(* IEC 61131-3 sources: 2026_Projet_YGO_ExcavatriceDragage/CODE/SIMULATION/PLC_TESTS/CORE, 4 files *)

(* ---- FB_TestSequencer.st ---- *)
FUNCTION_BLOCK FB_TestSequencer
VAR_INPUT
    Start       : BOOL;              // Front : lance à FirstStepId
    Abort       : BOOL;              // Niveau : arrêt immédiat propre
    FirstStepId : INT;               // Run all = 1er SETUP ; run one = FirstStep du case visé
END_VAR
VAR_IN_OUT                           // 🔗 zéro copie
    StepTable      : ARRAY[1..GVL_PLC_Tests_Const.MaxSteps]      OF ST_TestStepConfig;
    CheckTable     : ARRAY[1..GVL_PLC_Tests_Const.MaxChecks]     OF ST_TestCheckConfig;
    CaseTable      : ARRAY[1..GVL_PLC_Tests_Const.MaxTestCases]  OF ST_TestCaseConfig;
    InvariantTable : ARRAY[1..GVL_PLC_Tests_Const.MaxInvariants] OF ST_TestInvariantConfig;
    ProbeBool      : ARRAY[1..GVL_PLC_Tests_Const.MaxProbeBool]  OF BOOL;
    ProbeDint      : ARRAY[1..GVL_PLC_Tests_Const.MaxProbeDint]  OF DINT;
    ProbeReal      : ARRAY[1..GVL_PLC_Tests_Const.MaxProbeReal]  OF REAL;
    Report         : ST_TestSuiteReport;
END_VAR
VAR_OUTPUT
    Busy                : BOOL;
    Done                : BOOL;
    AnyFailed           : BOOL;
    ConfigError         : BOOL;      // 🔒 Table invalide -> refus de lancer
    ConfigErrorStepId   : INT;
    ConfigErrorCheckIdx : INT;
    CurrentStepId       : INT;
    ActiveStimulusId    : INT;       // ⚡ consommé par le domaine
    StepElapsed         : TIME;      // Pour l'IHM
END_VAR
VAR
    StartTrig           : R_TRIG;
    StepTimer           : TON;
    DwellTimer          : TON;
    Checks              : ARRAY[1..GVL_PLC_Tests_Const.MaxChecksPerStep] OF FB_TestCheck;
    InvChecks           : ARRAY[1..GVL_PLC_Tests_Const.MaxInvariants]    OF FB_TestCheck;
    InvArmed            : ARRAY[1..GVL_PLC_Tests_Const.MaxInvariants]    OF BOOL;

    // Variables de contrôle internes
    StepStarted         : BOOL;
    CurrentCaseId       : INT;
    Idx                 : INT;
    Jdx                 : INT;
    Kdx                 : INT;
    Valid               : BOOL;

    // 🔧 REX : locaux remontés depuis des blocs VAR imbriqués dans le corps
    AllChecksPassed     : BOOL;
    AnyCheckFailed      : BOOL;
    FailedCheckIdxLocal : INT;
    FailReasonLocal     : E_TestFailReason;
    ObsBoolLocal        : BOOL;
    ObsDintLocal        : DINT;
    ObsRealLocal        : REAL;
    NeverDuringPassed   : BOOL;
    SuiteAllPassed      : BOOL;
    FirstFailedCase     : INT;
    CaseIdx             : INT;
    CaseStartStep       : INT;
    CaseStep            : INT;
    CaseOk              : BOOL;
    CaseExecuted        : BOOL;
    CaseFailedStep      : INT;
    CaseDuration        : TIME;
    CaseFailReason      : E_TestFailReason;
END_VAR
// === IMPLEMENTATION ===
StartTrig(CLK := Start);

// 1. Validation de la configuration sur front de Start
IF StartTrig.Q THEN
    ConfigError := FALSE;
    ConfigErrorStepId := 0;
    ConfigErrorCheckIdx := 0;

    // Validation des étapes
    FOR Idx := 1 TO GVL_PLC_Tests_Const.MaxSteps DO
        IF StepTable[Idx].CaseId > 0 THEN
            // Vérification des NextOn
            IF StepTable[Idx].NextOnPass < 0 OR StepTable[Idx].NextOnPass > GVL_PLC_Tests_Const.MaxSteps THEN
                ConfigError := TRUE;
                ConfigErrorStepId := Idx;
            ELSIF StepTable[Idx].NextOnFail < 0 OR StepTable[Idx].NextOnFail > GVL_PLC_Tests_Const.MaxSteps THEN
                ConfigError := TRUE;
                ConfigErrorStepId := Idx;
            END_IF;

            // Vérification du Timeout
            IF StepTable[Idx].TimeoutPT <= T#0s THEN
                // Sauf si tous les checks de cette étape sont NEVER_DURING, mais restons stricts : TimeoutPT requis
                ConfigError := TRUE;
                ConfigErrorStepId := Idx;
            END_IF;

            // Vérification des Checks indexés par l'étape
            FOR Jdx := 1 TO GVL_PLC_Tests_Const.MaxChecksPerStep DO
                Kdx := StepTable[Idx].CheckIdx[Jdx];
                IF Kdx > 0 THEN
                    IF Kdx > GVL_PLC_Tests_Const.MaxChecks THEN
                        ConfigError := TRUE;
                        ConfigErrorStepId := Idx;
                        ConfigErrorCheckIdx := Kdx;
                    ELSE
                        // Validation de la sonde associée au check
                        CASE CheckTable[Kdx].Kind OF
                            E_TestCheckKind.BOOL_EQUAL, E_TestCheckKind.BOOL_RISING, E_TestCheckKind.BOOL_FALLING:
                                IF CheckTable[Kdx].ProbeIdx < 1 OR CheckTable[Kdx].ProbeIdx > GVL_PLC_Tests_Const.MaxProbeBool THEN
                                    ConfigError := TRUE;
                                    ConfigErrorStepId := Idx;
                                    ConfigErrorCheckIdx := Kdx;
                                END_IF;
                            E_TestCheckKind.DINT_EQUAL, E_TestCheckKind.DINT_NOT_EQUAL, E_TestCheckKind.DINT_IN_RANGE,
                            E_TestCheckKind.WORD_MASK_ALL, E_TestCheckKind.WORD_MASK_ANY, E_TestCheckKind.WORD_MASK_NONE:
                                IF CheckTable[Kdx].ProbeIdx < 1 OR CheckTable[Kdx].ProbeIdx > GVL_PLC_Tests_Const.MaxProbeDint THEN
                                    ConfigError := TRUE;
                                    ConfigErrorStepId := Idx;
                                    ConfigErrorCheckIdx := Kdx;
                                END_IF;
                            E_TestCheckKind.REAL_IN_RANGE:
                                IF CheckTable[Kdx].ProbeIdx < 1 OR CheckTable[Kdx].ProbeIdx > GVL_PLC_Tests_Const.MaxProbeReal THEN
                                    ConfigError := TRUE;
                                    ConfigErrorStepId := Idx;
                                    ConfigErrorCheckIdx := Kdx;
                                END_IF;
                        END_CASE;
                    END_IF;
                END_IF;
            END_FOR;
        END_IF;
    END_FOR;

    // Si erreur de config, on bloque le démarrage
    IF ConfigError THEN
        RETURN;
    END_IF;
END_IF;

// 2. Abort (Niveau, priorité absolue)
IF Abort THEN
    IF Busy THEN
        Report.InProgress := FALSE;
        Report.Aborted := TRUE;
        Report.AnyFailed := TRUE;

        // Enregistrement de l'échec de l'étape courante
        IF CurrentStepId >= 1 AND CurrentStepId <= GVL_PLC_Tests_Const.MaxSteps THEN
            Report.Steps[CurrentStepId].Executed := TRUE;
            Report.Steps[CurrentStepId].Passed := FALSE;
            Report.Steps[CurrentStepId].FailReason := E_TestFailReason.FAIL_ABORTED;
            Report.Steps[CurrentStepId].Duration := StepElapsed;
        END_IF;

        // Échec du cas de test en cours
        IF CurrentCaseId >= 1 AND CurrentCaseId <= GVL_PLC_Tests_Const.MaxTestCases THEN
            Report.Cases[CurrentCaseId].Ok := FALSE;
            Report.Cases[CurrentCaseId].FailReason := E_TestFailReason.FAIL_ABORTED;
        END_IF;

        Busy := FALSE;
        Done := TRUE;
        AnyFailed := TRUE;
    END_IF;
    ActiveStimulusId := 0;
    StepStarted := FALSE;
    RETURN;
END_IF;

// 3. Démarrage de la suite
IF StartTrig.Q AND NOT ConfigError THEN
    Busy := TRUE;
    Done := FALSE;
    AnyFailed := FALSE;
    CurrentStepId := FirstStepId;
    StepStarted := FALSE;

    // RAZ Rapport
    Report.InProgress := TRUE;
    Report.AllPassed := FALSE;
    Report.AnyFailed := FALSE;
    Report.Aborted := FALSE;
    Report.FailedTestCase := 0;
    Report.CurrentStepId := FirstStepId;
    IF CurrentStepId >= 1 AND CurrentStepId <= GVL_PLC_Tests_Const.MaxSteps THEN
        Report.CurrentCaseId := StepTable[CurrentStepId].CaseId;
    ELSE
        Report.CurrentCaseId := 0;
    END_IF;
    Report.Duration := T#0s;
    Report.RunCounter := Report.RunCounter + 1;

    FOR Idx := 1 TO GVL_PLC_Tests_Const.MaxSteps DO
        Report.Steps[Idx].Executed := FALSE;
        Report.Steps[Idx].Passed := FALSE;
        Report.Steps[Idx].FailReason := E_TestFailReason.FAIL_NONE;
        Report.Steps[Idx].FailedCheckIdx := 0;
        Report.Steps[Idx].FailedInvariantId := 0;
        Report.Steps[Idx].Duration := T#0s;
    END_FOR;

    FOR Idx := 1 TO GVL_PLC_Tests_Const.MaxTestCases DO
        Report.Cases[Idx].Executed := FALSE;
        Report.Cases[Idx].Ok := FALSE;
        Report.Cases[Idx].FailedStepId := 0;
        Report.Cases[Idx].FailReason := E_TestFailReason.FAIL_NONE;
        Report.Cases[Idx].Duration := T#0s;
    END_FOR;

    // RAZ Invariants
    FOR Idx := 1 TO GVL_PLC_Tests_Const.MaxInvariants DO
        InvArmed[Idx] := FALSE;
    END_FOR;
END_IF;

// 4. Moteur d'exécution principal
IF Busy THEN
    // Incrément de la durée globale du run
    Report.Duration := Report.Duration + UDINT_TO_TIME(INT_TO_UDINT(GVL_PLC_Tests_Const.TaskCycleMs));

    // Vérification des bornes de l'étape courante
    IF CurrentStepId < 1 OR CurrentStepId > GVL_PLC_Tests_Const.MaxSteps THEN
        Busy := FALSE;
        Done := TRUE;
        ActiveStimulusId := 0;
        RETURN;
    END_IF;

    CurrentCaseId := StepTable[CurrentStepId].CaseId;
    ActiveStimulusId := StepTable[CurrentStepId].StimulusId;
    Report.CurrentStepId := CurrentStepId;
    Report.CurrentCaseId := CurrentCaseId;

    IF NOT StepStarted THEN
        StepStarted := TRUE;
        StepElapsed := T#0s;
        DwellTimer(IN := FALSE);
        StepTimer(IN := FALSE);

        // Gestion de l'armement/désarmement des invariants
        FOR Idx := 1 TO GVL_PLC_Tests_Const.MaxInvariants DO
            IF InvariantTable[Idx].ArmAtStepId = CurrentStepId THEN
                InvArmed[Idx] := TRUE;
            END_IF;
            IF InvariantTable[Idx].DisarmAtStepId = CurrentStepId THEN
                InvArmed[Idx] := FALSE;
            END_IF;
        END_FOR;
    END_IF;

    // Incrément de la durée de l'étape courante
    StepElapsed := StepElapsed + UDINT_TO_TIME(INT_TO_UDINT(GVL_PLC_Tests_Const.TaskCycleMs));

    // 4.1 Évaluation des invariants actifs
    FOR Idx := 1 TO GVL_PLC_Tests_Const.MaxInvariants DO
        IF InvArmed[Idx] THEN
            InvChecks[Idx](Config := InvariantTable[Idx].Check, Evaluate := TRUE, ProbeBool := ProbeBool, ProbeDint := ProbeDint, ProbeReal := ProbeReal);
            IF InvChecks[Idx].Failed THEN
                // Violation d'invariant -> Transition en échec immédiat
                Report.Steps[CurrentStepId].Executed := TRUE;
                Report.Steps[CurrentStepId].Passed := FALSE;
                Report.Steps[CurrentStepId].FailReason := E_TestFailReason.FAIL_INVARIANT;
                Report.Steps[CurrentStepId].FailedInvariantId := Idx;
                Report.Steps[CurrentStepId].Duration := StepElapsed;
                Report.Steps[CurrentStepId].ObservedBool := InvChecks[Idx].ObservedBool;
                Report.Steps[CurrentStepId].ObservedDint := InvChecks[Idx].ObservedDint;
                Report.Steps[CurrentStepId].ObservedReal := InvChecks[Idx].ObservedReal;

                // Désactivation de l'évaluation
                InvChecks[Idx](Config := InvariantTable[Idx].Check, Evaluate := FALSE, ProbeBool := ProbeBool, ProbeDint := ProbeDint, ProbeReal := ProbeReal);

                // Transition
                IF StepTable[CurrentStepId].FailAction = E_TestFailAction.FAIL_ABORT_SUITE THEN
                    Busy := FALSE;
                    Done := TRUE;
                    AnyFailed := TRUE;
                    ActiveStimulusId := 0;
                ELSE
                    CurrentStepId := StepTable[CurrentStepId].NextOnFail;
                    StepStarted := FALSE;
                END_IF;
                RETURN;
            END_IF;
        END_IF;
    END_FOR;

    // 4.2 Gestion de la temporisation de Dwell
    DwellTimer(IN := TRUE, PT := StepTable[CurrentStepId].DwellPT);
    IF NOT DwellTimer.Q THEN
        // En attente du Dwell, pas d'évaluation des checks d'étape
        FOR Jdx := 1 TO GVL_PLC_Tests_Const.MaxChecksPerStep DO
            Checks[Jdx](Evaluate := FALSE, ProbeBool := ProbeBool, ProbeDint := ProbeDint, ProbeReal := ProbeReal);
        END_FOR;
        RETURN;
    END_IF;

    // 4.3 Évaluation des checks d'étape
    AllChecksPassed     := TRUE;
    AnyCheckFailed      := FALSE;
    FailedCheckIdxLocal := 0;
    FailReasonLocal     := E_TestFailReason.FAIL_NONE;
    ObsBoolLocal        := FALSE;
    ObsDintLocal        := 0;
    ObsRealLocal        := 0.0;

    FOR Jdx := 1 TO GVL_PLC_Tests_Const.MaxChecksPerStep DO
        Kdx := StepTable[CurrentStepId].CheckIdx[Jdx];
        IF Kdx > 0 THEN
            Checks[Jdx](Config := CheckTable[Kdx], Evaluate := TRUE, ProbeBool := ProbeBool, ProbeDint := ProbeDint, ProbeReal := ProbeReal);

            IF Checks[Jdx].Failed THEN
                AnyCheckFailed := TRUE;
                FailedCheckIdxLocal := Kdx;
                FailReasonLocal := Checks[Jdx].FailReason;
                ObsBoolLocal := Checks[Jdx].ObservedBool;
                ObsDintLocal := Checks[Jdx].ObservedDint;
                ObsRealLocal := Checks[Jdx].ObservedReal;
            ELSIF Checks[Jdx].Pending THEN
                AllChecksPassed := FALSE;
            END_IF;
        END_IF;
    END_FOR;

    // 4.4 Prise de verdict
    IF AnyCheckFailed THEN
        // Échec sur un check d'étape
        Report.Steps[CurrentStepId].Executed := TRUE;
        Report.Steps[CurrentStepId].Passed := FALSE;
        Report.Steps[CurrentStepId].FailReason := FailReasonLocal;
        Report.Steps[CurrentStepId].FailedCheckIdx := FailedCheckIdxLocal;
        Report.Steps[CurrentStepId].Duration := StepElapsed;
        Report.Steps[CurrentStepId].ObservedBool := ObsBoolLocal;
        Report.Steps[CurrentStepId].ObservedDint := ObsDintLocal;
        Report.Steps[CurrentStepId].ObservedReal := ObsRealLocal;

        // Reset checks
        FOR Jdx := 1 TO GVL_PLC_Tests_Const.MaxChecksPerStep DO
            Checks[Jdx](Evaluate := FALSE, ProbeBool := ProbeBool, ProbeDint := ProbeDint, ProbeReal := ProbeReal);
        END_FOR;

        IF StepTable[CurrentStepId].FailAction = E_TestFailAction.FAIL_ABORT_SUITE THEN
            Busy := FALSE;
            Done := TRUE;
            AnyFailed := TRUE;
            ActiveStimulusId := 0;
        ELSE
            CurrentStepId := StepTable[CurrentStepId].NextOnFail;
            StepStarted := FALSE;
        END_IF;
        RETURN;
    END_IF;

    StepTimer(IN := TRUE, PT := StepTable[CurrentStepId].TimeoutPT);

    IF AllChecksPassed THEN
        // Succès précoce (vérification MinPT)
        IF StepElapsed < StepTable[CurrentStepId].MinPT THEN
            // Réaction trop rapide = Échec
            Report.Steps[CurrentStepId].Executed := TRUE;
            Report.Steps[CurrentStepId].Passed := FALSE;
            Report.Steps[CurrentStepId].FailReason := E_TestFailReason.FAIL_WINDOW_EARLY;
            Report.Steps[CurrentStepId].Duration := StepElapsed;

            // Reset checks
            FOR Jdx := 1 TO GVL_PLC_Tests_Const.MaxChecksPerStep DO
                Checks[Jdx](Evaluate := FALSE, ProbeBool := ProbeBool, ProbeDint := ProbeDint, ProbeReal := ProbeReal);
            END_FOR;

            IF StepTable[CurrentStepId].FailAction = E_TestFailAction.FAIL_ABORT_SUITE THEN
                Busy := FALSE;
                Done := TRUE;
                AnyFailed := TRUE;
                ActiveStimulusId := 0;
            ELSE
                CurrentStepId := StepTable[CurrentStepId].NextOnFail;
                StepStarted := FALSE;
            END_IF;
        ELSE
            // Validation étape OK
            Report.Steps[CurrentStepId].Executed := TRUE;
            Report.Steps[CurrentStepId].Passed := TRUE;
            Report.Steps[CurrentStepId].Duration := StepElapsed;

            // Prendre snapshot du premier check s'il existe
            IF StepTable[CurrentStepId].CheckIdx[1] > 0 THEN
                Report.Steps[CurrentStepId].ObservedBool := Checks[1].ObservedBool;
                Report.Steps[CurrentStepId].ObservedDint := Checks[1].ObservedDint;
                Report.Steps[CurrentStepId].ObservedReal := Checks[1].ObservedReal;
            END_IF;

            // Reset checks
            FOR Jdx := 1 TO GVL_PLC_Tests_Const.MaxChecksPerStep DO
                Checks[Jdx](Evaluate := FALSE, ProbeBool := ProbeBool, ProbeDint := ProbeDint, ProbeReal := ProbeReal);
            END_FOR;

            CurrentStepId := StepTable[CurrentStepId].NextOnPass;
            StepStarted := FALSE;
        END_IF;
        RETURN;
    END_IF;

    // Gestion du timeout d'étape
    IF StepTimer.Q THEN
        // Si timeout expiré, vérifions si des checks NEVER_DURING sont en attente
        NeverDuringPassed := TRUE;
        FOR Jdx := 1 TO GVL_PLC_Tests_Const.MaxChecksPerStep DO
            Kdx := StepTable[CurrentStepId].CheckIdx[Jdx];
            IF Kdx > 0 THEN
                IF CheckTable[Kdx].Mode = E_TestCheckMode.CHECK_NEVER_DURING THEN
                    // Jamais violé pendant toute la fenêtre
                    Checks[Jdx](Evaluate := FALSE, ProbeBool := ProbeBool, ProbeDint := ProbeDint, ProbeReal := ProbeReal);
                ELSE
                    // Les autres modes auraient dû passer avant le timeout
                    NeverDuringPassed := FALSE;
                END_IF;
            END_IF;
        END_FOR;

        IF NeverDuringPassed THEN
            // Succès par non-violation
            Report.Steps[CurrentStepId].Executed := TRUE;
            Report.Steps[CurrentStepId].Passed := TRUE;
            Report.Steps[CurrentStepId].Duration := StepElapsed;

            CurrentStepId := StepTable[CurrentStepId].NextOnPass;
            StepStarted := FALSE;
        ELSE
            // Timeout classique de l'étape
            Report.Steps[CurrentStepId].Executed := TRUE;
            Report.Steps[CurrentStepId].Passed := FALSE;
            Report.Steps[CurrentStepId].FailReason := E_TestFailReason.FAIL_TIMEOUT;
            Report.Steps[CurrentStepId].Duration := StepElapsed;

            IF StepTable[CurrentStepId].FailAction = E_TestFailAction.FAIL_ABORT_SUITE THEN
                Busy := FALSE;
                Done := TRUE;
                AnyFailed := TRUE;
                ActiveStimulusId := 0;
            ELSE
                CurrentStepId := StepTable[CurrentStepId].NextOnFail;
                StepStarted := FALSE;
            END_IF;
        END_IF;

        // Reset checks
        FOR Jdx := 1 TO GVL_PLC_Tests_Const.MaxChecksPerStep DO
            Checks[Jdx](Evaluate := FALSE, ProbeBool := ProbeBool, ProbeDint := ProbeDint, ProbeReal := ProbeReal);
        END_FOR;
    END_IF;
END_IF;

// 5. Agrégation des résultats en fin de suite (CurrentStepId = 0)
IF Busy AND CurrentStepId = 0 THEN
    Busy := FALSE;
    Done := TRUE;
    ActiveStimulusId := 0;
    Report.InProgress := FALSE;

    // Agrégation des cas de test
    SuiteAllPassed  := TRUE;
    FirstFailedCase := 0;

    FOR CaseIdx := 1 TO GVL_PLC_Tests_Const.MaxTestCases DO
        CaseStartStep := CaseTable[CaseIdx].FirstStep;
        IF CaseStartStep > 0 THEN
            CaseOk := TRUE;
            CaseExecuted := FALSE;
            CaseFailedStep := 0;
            CaseDuration := T#0s;
            CaseFailReason := E_TestFailReason.FAIL_NONE;

            // Parcourir la chaîne d'étapes à partir de FirstStep
            CaseStep := CaseStartStep;
            WHILE CaseStep > 0 AND StepTable[CaseStep].CaseId = CaseIdx DO
                IF Report.Steps[CaseStep].Executed THEN
                    CaseExecuted := TRUE;
                    CaseDuration := CaseDuration + Report.Steps[CaseStep].Duration;
                    IF NOT Report.Steps[CaseStep].Passed THEN
                        CaseOk := FALSE;
                        CaseFailedStep := CaseStep;
                        CaseFailReason := Report.Steps[CaseStep].FailReason;
                    END_IF;
                END_IF;

                // Suivre NextOnPass ou NextOnFail selon l'exécution réelle
                IF Report.Steps[CaseStep].Executed AND NOT Report.Steps[CaseStep].Passed THEN
                    CaseStep := StepTable[CaseStep].NextOnFail;
                ELSE
                    CaseStep := StepTable[CaseStep].NextOnPass;
                END_IF;
            END_WHILE;

            Report.Cases[CaseIdx].Executed := CaseExecuted;
            Report.Cases[CaseIdx].Ok := CaseExecuted AND CaseOk;
            Report.Cases[CaseIdx].FailedStepId := CaseFailedStep;
            Report.Cases[CaseIdx].FailReason := CaseFailReason;
            Report.Cases[CaseIdx].Duration := CaseDuration;

            IF CaseExecuted AND NOT CaseOk THEN
                SuiteAllPassed := FALSE;
                IF FirstFailedCase = 0 THEN
                    FirstFailedCase := CaseIdx;
                END_IF;
            END_IF;
        END_IF;
    END_FOR;

    Report.AllPassed := SuiteAllPassed;
    Report.AnyFailed := NOT SuiteAllPassed;
    Report.FailedTestCase := FirstFailedCase;
    AnyFailed := NOT SuiteAllPassed;
END_IF;

(* ---- FB_TranslationTestCleanup.st ---- *)
// ═══════════════════════════════════════════════════════════════
// 🧪 FB_TranslationTestCleanup — Neutralité Translation M3
// ───────────────────────────────────────────────────────────────
// 🎯 Responsabilité UNIQUE : porter le vecteur d'état NEUTRE complet
//    (tous les overrides M3 relâchés, instance isolée FB_Translation
//    au repos). Source de vérité UNIQUE de "neutre" — appelée depuis
//    le fichier suite (SUITE_TRANSLATION/FB_TranslationValidation.st)
//    à la fois dans le CASE stimulus (StimulusId=0) ET, en garantie
//    structurelle indépendante, sur tout chemin où la suite n'est pas
//    Busy (ceinture + bretelles, AF_Partie-14 §7.3.2).
// 🚫 Ne force JAMAIS une sortie de commande calculée — uniquement les
//    surcharges capteurs amont (GVL_PLC_Tests.OverrideM3*) et les
//    entrées de l'instance de test isolée.
// ═══════════════════════════════════════════════════════════════

FUNCTION_BLOCK PUBLIC FB_TranslationTestCleanup
VAR_INPUT
    Apply : BOOL; // TRUE = force la neutralité maintenant
END_VAR
VAR_OUTPUT
    OverrideAtTremie          : BOOL;
    OverrideBrakeStuckOpen    : BOOL;
    OverridePhantomFreq       : BOOL;
    OverrideSensorsWordActive : BOOL;
    UnderTestDirection        : INT;
    UnderTestStartStop        : BOOL;
    UnderTestSlowdownSensor   : BOOL;
    NeutralConfirmed          : BOOL; // TRUE dès que la neutralité a été appliquée ce scan
END_VAR
// === IMPLEMENTATION ===
IF Apply THEN
    OverrideAtTremie := FALSE;
    OverrideBrakeStuckOpen := FALSE;
    OverridePhantomFreq := FALSE;
    OverrideSensorsWordActive := FALSE;
    UnderTestDirection := 0;
    UnderTestStartStop := FALSE;
    UnderTestSlowdownSensor := FALSE;
    NeutralConfirmed := TRUE;
ELSE
    NeutralConfirmed := FALSE;
END_IF;

(* ---- FB_TranslationTestFixture.st ---- *)
// ═══════════════════════════════════════════════════════════════
// 🧪 FB_TranslationTestFixture — Précondition Translation M3
// ───────────────────────────────────────────────────────────────
// 🎯 Responsabilité UNIQUE : décider si un Start est recevable
//    (Niveaux 1/2 de la défense en profondeur, AF_Partie-14 §7.3.3) :
//    simulation active + aucune E/S M3 recâblée réelle. Ne fait AUCUNE
//    attente d'état sain (ça reste la responsabilité de l'étape SETUP
//    de chaque cas, via FB_TranslationStepExecutor — §7.3.5).
// 🔒 Un refus ici est TOUJOURS explicite (PRECONDITION_FAILED),
//    jamais un silence (audit v1.0 C3).
// ═══════════════════════════════════════════════════════════════

FUNCTION_BLOCK PUBLIC FB_TranslationTestFixture
VAR_INPUT
    CheckRequested        : BOOL; // Front : nouvelle vérification demandée (sur Start suite)
    SimulationModeActive  : BOOL;
    SimGateOk             : BOOL; // Niveau 2 : aucune E/S M3 (*IsReal) incompatible
END_VAR
VAR_OUTPUT
    FixturePassed  : BOOL;
    FixtureFailed  : BOOL;
    FailReason     : STRING(120);
END_VAR
VAR
    CheckTrig : R_TRIG;
END_VAR
// === IMPLEMENTATION ===
CheckTrig(CLK := CheckRequested);

IF CheckTrig.Q THEN
    IF NOT SimulationModeActive THEN
        FixturePassed := FALSE;
        FixtureFailed := TRUE;
        FailReason := 'Simulation non active (GVL_Simulation.SimulationModeActive=FALSE)';
    ELSIF NOT SimGateOk THEN
        FixturePassed := FALSE;
        FixtureFailed := TRUE;
        FailReason := 'E/S M3 recablees reelles (*IsReal) incompatibles avec le banc de test';
    ELSE
        FixturePassed := TRUE;
        FixtureFailed := FALSE;
        FailReason := '';
    END_IF;
END_IF;

(* ---- FB_TranslationTestRuntime.st ---- *)
// ═══════════════════════════════════════════════════════════════
// 🧪 FB_TranslationTestRuntime — Cycle de vie protégé Translation M3
// ───────────────────────────────────────────────────────────────
// 🎯 Responsabilité UNIQUE : posséder le lifecycle atomique du run :
//    IDLE → RUN → CLEANUP → WAIT_NEUTRAL → VERIFY → TERMINAL.
// 🔒 Aucun terminal n'est publié avant neutralité confirmée.
// ═══════════════════════════════════════════════════════════════

FUNCTION_BLOCK PUBLIC FB_TranslationTestRuntime
VAR_INPUT
    Start   : BOOL;
    Abort   : BOOL;
    CaseId  : INT;
    PlanConfigError         : BOOL;
    PlanConfigErrorStepId   : INT;
    PlanConfigErrorCheckIdx : INT;
    PlanConfigErrorMessage  : STRING(160);
    SimulationModeActive    : BOOL;
    SimGateOk               : BOOL;
    NeutralConfirmed        : BOOL; // Neutralité réellement appliquée au scan précédent
    WatchdogLimitMs         : DINT := 180000; // Paramétrable pour autotest du framework
    CleanupTimeoutScans     : INT := 20;      // Délai max de confirmation du neutre
END_VAR
VAR_IN_OUT
    StepTable  : ARRAY[1..GVL_PLC_Tests_Const.MaxSteps]      OF ST_TestStepConfig;
    CheckTable : ARRAY[1..GVL_PLC_Tests_Const.MaxChecks]     OF ST_TestCheckConfig;
    CaseTable  : ARRAY[1..GVL_PLC_Tests_Const.MaxTestCases]  OF ST_TestCaseConfig;
    ProbeBool  : ARRAY[1..GVL_PLC_Tests_Const.MaxProbeBool]  OF BOOL;
    ProbeDint  : ARRAY[1..GVL_PLC_Tests_Const.MaxProbeDint]  OF DINT;
    ProbeReal  : ARRAY[1..GVL_PLC_Tests_Const.MaxProbeReal]  OF REAL;
    Report     : ST_TestSuiteReport;
    Result     : ST_TranslationTestResult;
END_VAR
VAR_OUTPUT
    Busy                : BOOL;
    Done                : BOOL;
    AnyFailed           : BOOL;
    ActiveStimulusId    : INT;
    StepElapsed         : TIME;
    TerminalState       : E_TestTerminalState;
    ConfigError         : BOOL;
    ConfigErrorStepId   : INT;
    ConfigErrorCheckIdx : INT;
    ErrorCode           : INT;
    ErrorMessage        : STRING(160);
    StartRejected       : BOOL; // Impulsion : Start reçu hors IDLE/TERMINAL
    CleanupRequest      : BOOL; // Niveau : imposer le vecteur neutre complet
END_VAR
VAR CONSTANT
    RuntimeIdle        : INT := 0;
    RuntimeRun         : INT := 10;
    RuntimeCleanup     : INT := 20;
    RuntimeWaitNeutral : INT := 30;
    RuntimeVerify      : INT := 40;
    RuntimeTerminal    : INT := 50;
END_VAR
VAR
    instFixture   : FB_TranslationTestFixture;
    instExecutor  : FB_TranslationStepExecutor;
    instFinalizer : FB_TranslationReportFinalizer;
    StartTrig     : R_TRIG;
    RuntimeState  : INT := 0;
    ExecutorStart : BOOL;
    ExecutorAbort : BOOL;
    RunStartPulse : BOOL;
    FinalizePulse : BOOL;
    PendingTerminalState : E_TestTerminalState;
    PendingErrorCode     : INT;
    PendingErrorMessage  : STRING(160);
    SuiteElapsed         : TIME;
    NeutralWaitScans     : INT;
    CleanupElapsedScans  : INT;
END_VAR
// === IMPLEMENTATION ===
StartTrig(CLK := Start);
StartRejected := FALSE;
ExecutorStart := FALSE;
ExecutorAbort := FALSE;
RunStartPulse := FALSE;
FinalizePulse := FALSE;
CleanupRequest := (RuntimeState = RuntimeCleanup)
               OR (RuntimeState = RuntimeWaitNeutral)
               OR (RuntimeState = RuntimeVerify);

// 🎮 Un Start pendant un run/cleanup est refusé sans modifier le run actif.
IF StartTrig.Q AND RuntimeState <> RuntimeIdle AND RuntimeState <> RuntimeTerminal THEN
    StartRejected := TRUE;
END_IF;

// 🚪 Fixture appelée CHAQUE scan : son R_TRIG interne est ainsi toujours réarmé.
instFixture(CheckRequested := StartTrig.Q,
            SimulationModeActive := SimulationModeActive,
            SimGateOk := SimGateOk);

// 🟢 Nouveau run accepté depuis IDLE ou TERMINAL.
IF StartTrig.Q AND (RuntimeState = RuntimeIdle OR RuntimeState = RuntimeTerminal) THEN
    RunStartPulse := TRUE;
    Done := FALSE;
    SuiteElapsed := T#0s;
    NeutralWaitScans := 0;
    CleanupElapsedScans := 0;
    PendingTerminalState := E_TestTerminalState.TEST_TERMINAL_NONE;
    PendingErrorCode := 0;
    PendingErrorMessage := '';

    IF PlanConfigError THEN
        PendingTerminalState := E_TestTerminalState.TEST_TERMINAL_CONFIG_ERROR;
        PendingErrorCode := 1002;
        PendingErrorMessage := CONCAT('Table invalide : ', PlanConfigErrorMessage);
        RuntimeState := RuntimeCleanup;
    ELSIF CaseId < 0 OR CaseId > 6 THEN
        PendingTerminalState := E_TestTerminalState.TEST_TERMINAL_CONFIG_ERROR;
        PendingErrorCode := 1001;
        PendingErrorMessage := 'CaseId invalide (attendu 0..6)';
        RuntimeState := RuntimeCleanup;
    ELSIF instFixture.FixtureFailed THEN
        PendingTerminalState := E_TestTerminalState.TEST_TERMINAL_PRECONDITION_FAILED;
        PendingErrorCode := 1010;
        PendingErrorMessage := CONCAT('PRECONDITION_FAILED : ', instFixture.FailReason);
        RuntimeState := RuntimeCleanup;
    ELSE
        ExecutorStart := TRUE;
        RuntimeState := RuntimeRun;
    END_IF;
END_IF;

// 🛡️ Causes de sortie du RUN : watchdog > gate perdue > abort opérateur.
IF RuntimeState = RuntimeRun THEN
    SuiteElapsed := SuiteElapsed + UDINT_TO_TIME(INT_TO_UDINT(GVL_PLC_Tests_Const.TaskCycleMs));
    IF SuiteElapsed >= DINT_TO_TIME(WatchdogLimitMs) THEN
        ExecutorAbort := TRUE;
        PendingTerminalState := E_TestTerminalState.TEST_TERMINAL_WATCHDOG_TIMEOUT;
        PendingErrorCode := 1020;
        PendingErrorMessage := 'Watchdog suite Translation expire';
    ELSIF NOT SimulationModeActive OR NOT SimGateOk THEN
        ExecutorAbort := TRUE;
        PendingTerminalState := E_TestTerminalState.TEST_TERMINAL_PRECONDITION_FAILED;
        PendingErrorCode := 1011;
        PendingErrorMessage := 'Gate Translation perdue pendant le run';
    ELSIF Abort THEN
        ExecutorAbort := TRUE;
        PendingTerminalState := E_TestTerminalState.TEST_TERMINAL_ABORTED;
        PendingErrorCode := 1030;
        PendingErrorMessage := 'Abandon operateur';
    END_IF;
END_IF;

// 🪜 L'exécuteur ne possède que les étapes, jamais le terminal public.
instExecutor(
    Start := ExecutorStart,
    Abort := ExecutorAbort,
    CaseId := CaseId,
    StepTable := StepTable,
    CheckTable := CheckTable,
    CaseTable := CaseTable,
    ProbeBool := ProbeBool,
    ProbeDint := ProbeDint,
    ProbeReal := ProbeReal
);

IF RuntimeState = RuntimeRun AND instExecutor.RunDone THEN
    IF PendingTerminalState = E_TestTerminalState.TEST_TERMINAL_NONE THEN
        PendingTerminalState := instExecutor.TerminalState;
        IF instExecutor.ConfigError THEN
            PendingErrorCode := 1003;
            PendingErrorMessage := 'Garde-fou runtime : transition invalide';
        END_IF;
    END_IF;
    RuntimeState := RuntimeCleanup;
    NeutralWaitScans := 0;
END_IF;

// 🧹 Tous les chemins imposent au moins deux scans complets au neutre.
IF RuntimeState = RuntimeCleanup THEN
    CleanupRequest := TRUE;
    NeutralWaitScans := 0;
    CleanupElapsedScans := 0;
    RuntimeState := RuntimeWaitNeutral;
ELSIF RuntimeState = RuntimeWaitNeutral THEN
    CleanupRequest := TRUE;
    NeutralWaitScans := NeutralWaitScans + 1;
    CleanupElapsedScans := CleanupElapsedScans + 1;
    IF NeutralWaitScans >= 2 THEN
        RuntimeState := RuntimeVerify;
    END_IF;
ELSIF RuntimeState = RuntimeVerify THEN
    CleanupRequest := TRUE;
    CleanupElapsedScans := CleanupElapsedScans + 1;
    IF NeutralConfirmed THEN
        FinalizePulse := TRUE;
        RuntimeState := RuntimeTerminal;
        Done := TRUE;
    ELSIF CleanupElapsedScans >= CleanupTimeoutScans THEN
        PendingTerminalState := E_TestTerminalState.TEST_TERMINAL_CONFIG_ERROR;
        PendingErrorCode := 1040;
        PendingErrorMessage := 'Cleanup Translation non confirme';
        FinalizePulse := TRUE;
        RuntimeState := RuntimeTerminal;
        Done := TRUE;
    END_IF;
END_IF;

// 📊 Le rapport consomme directement chaque verdict, même consécutif.
instFinalizer(
    RunStart := RunStartPulse,
    RequestedCaseId := CaseId,
    Busy := (RuntimeState = RuntimeRun),
    StepVerdict := instExecutor.StepVerdict,
    StepId := instExecutor.VerdictStepId,
    StepCaseId := instExecutor.VerdictCaseId,
    StepPassed := instExecutor.VerdictPassed,
    StepFailReason := instExecutor.VerdictFailReason,
    StepFailedCheckIdx := instExecutor.VerdictFailedCheckIdx,
    StepDuration := instExecutor.VerdictDuration,
    StepObservedBool := instExecutor.VerdictObservedBool,
    StepObservedDint := instExecutor.VerdictObservedDint,
    StepObservedReal := instExecutor.VerdictObservedReal,
    Finalize := FinalizePulse,
    TerminalState := PendingTerminalState,
    ErrorCode := PendingErrorCode,
    ErrorMessage := PendingErrorMessage,
    StepTable := StepTable,
    CaseTable := CaseTable,
    Report := Report,
    Result := Result
);

// 📤 Publication : Busy inclut cleanup ; aucun stimulus métier hors RUN.
Busy := (RuntimeState = RuntimeRun)
     OR (RuntimeState = RuntimeCleanup)
     OR (RuntimeState = RuntimeWaitNeutral)
     OR (RuntimeState = RuntimeVerify);
IF RuntimeState = RuntimeRun THEN
    ActiveStimulusId := instExecutor.ActiveStimulusId;
ELSE
    ActiveStimulusId := 0;
END_IF;
StepElapsed := instExecutor.StepElapsed;
TerminalState := Result.TerminalState;
AnyFailed := Result.AnyFailed;
ConfigError := PlanConfigError OR instExecutor.ConfigError;
IF PlanConfigError THEN
    ConfigErrorStepId := PlanConfigErrorStepId;
    ConfigErrorCheckIdx := PlanConfigErrorCheckIdx;
ELSE
    ConfigErrorStepId := instExecutor.ConfigErrorStepId;
    ConfigErrorCheckIdx := 0;
END_IF;
ErrorCode := Result.ErrorCode;
ErrorMessage := Result.ErrorMessage;
